{attribute 'GeneratedUsingTerminal: EK1100-0000-0018'}
{attribute addProperty BoxType "EK1100-0000-0018"}
{attribute addProperty Id "Beckhoff_EP9xxxEK1122Beckhoff_EP9xxxEK1122_448E973C539A_0023_EP9224_1037_0017EP9224_1FC0878B2A_0015_EP9128_2021_0019EP9128_1FC0878B2A_0014_EP9128_1021_0019EP9128_1FC0878B2A_0012_EP9128_2021_0018EP9128_1FC0878B2A_0011_EP9128_1021_0018EP9128_1FC0878B2A_0009_EP9128_2021_0017EP9128_1FC0878B2A_0008_EP9128_1021_0017EP9128_1FC0878B2A_0006_EP9128_2021_0016EP9128_1FC0878B2A_0005_EP9128_1021_0016EP9128_1FC0878B2A_0003_EP9128_2020_0016EP9128_1FC0878B2A_0002_EP9128_1020_0016EP9128_1FC0878B2"}
{attribute addProperty CRC "960615833"}
{attribute addProperty Size "561"}
TYPE Beckhoff_EP9xxx_3941D599 EXTENDS EK1100_1FC0878B :
STRUCT
	{attribute addProperty Name "Beckhoff_EP9xxxEK1122"}
	{attribute addProperty PreviousPort "Beckhoff EP9xxx : B"}
	Beckhoff_EP9xxxEK1122 : Beckhoff_EP9xxxEK1122_448E973C;
	{attribute addProperty Name "A_0023_EP9224_1037_0017"}
	{attribute addProperty PreviousPort "Beckhoff EP9xxxEK1122 : C"}
	A_0023_EP9224_1037_0017 : EP9224_1FC0878B;
	{attribute addProperty Name "A_0015_EP9128_2021_0019"}
	{attribute addProperty PreviousPort "Beckhoff EP9xxxEK1122 : C"}
	A_0015_EP9128_2021_0019 : EP9128_1FC0878B;
	{attribute addProperty Name "A_0014_EP9128_1021_0019"}
	{attribute addProperty PreviousPort "Beckhoff EP9xxxEK1122 : C"}
	A_0014_EP9128_1021_0019 : EP9128_1FC0878B;
	{attribute addProperty Name "A_0012_EP9128_2021_0018"}
	{attribute addProperty PreviousPort "A_0014(EP9128-1021-0019) : C"}
	A_0012_EP9128_2021_0018 : EP9128_1FC0878B;
	{attribute addProperty Name "A_0011_EP9128_1021_0018"}
	{attribute addProperty PreviousPort "Beckhoff EP9xxxEK1122 : C"}
	A_0011_EP9128_1021_0018 : EP9128_1FC0878B;
	{attribute addProperty Name "A_0009_EP9128_2021_0017"}
	{attribute addProperty PreviousPort "A_0011(EP9128-1021-0018) : C"}
	A_0009_EP9128_2021_0017 : EP9128_1FC0878B;
	{attribute addProperty Name "A_0008_EP9128_1021_0017"}
	{attribute addProperty PreviousPort "Beckhoff EP9xxxEK1122 : C"}
	A_0008_EP9128_1021_0017 : EP9128_1FC0878B;
	{attribute addProperty Name "A_0006_EP9128_2021_0016"}
	{attribute addProperty PreviousPort "A_0008(EP9128-1021-0017) : C"}
	A_0006_EP9128_2021_0016 : EP9128_1FC0878B;
	{attribute addProperty Name "A_0005_EP9128_1021_0016"}
	{attribute addProperty PreviousPort "Beckhoff EP9xxxEK1122 : C"}
	A_0005_EP9128_1021_0016 : EP9128_1FC0878B;
	{attribute addProperty Name "A_0003_EP9128_2020_0016"}
	{attribute addProperty PreviousPort "A_0005(EP9128-1021-0016) : C"}
	A_0003_EP9128_2020_0016 : EP9128_1FC0878B;
	{attribute addProperty Name "A_0002_EP9128_1020_0016"}
	{attribute addProperty PreviousPort "Beckhoff EP9xxxEK1122 : C"}
	A_0002_EP9128_1020_0016 : EP9128_1FC0878B;
END_STRUCT
END_TYPE

(* stored: Version 1.2.0.0, ProductVersion 3.1.4024.9
   DUT Beckhoff_EP9xxx_3941D599: Id {6c9a42e3-7bad-4070-845c-b6dd057126c3} *)
